// TIA Portal V19 export
FUNCTION_BLOCK "FB20_ManageState"   // FB20, LAD
{ S7_Optimized_Access := 'TRUE' }
// stored: AutoNumber false, IsIECCheckEnabled true, MemoryReserve 100, SetENOAutomatically false
   VAR_INPUT
      xGlobalSafety { ExternalAccessible := 'False'; ExternalVisible := 'False'; ExternalWritable := 'False'} : Bool;
      xGlobalFault { ExternalAccessible := 'False'; ExternalVisible := 'False'; ExternalWritable := 'False'} : Bool;
      xInformation { ExternalAccessible := 'False'; ExternalVisible := 'False'; ExternalWritable := 'False'} : Bool;
   END_VAR
   VAR_OUTPUT
      nGlobalState { ExternalAccessible := 'False'; ExternalVisible := 'False'; ExternalWritable := 'False'} : Int;
      xSafetyState { ExternalAccessible := 'False'; ExternalVisible := 'False'; ExternalWritable := 'False'} : Bool;
   END_VAR
BEGIN

REGION Network 1: Safety fault
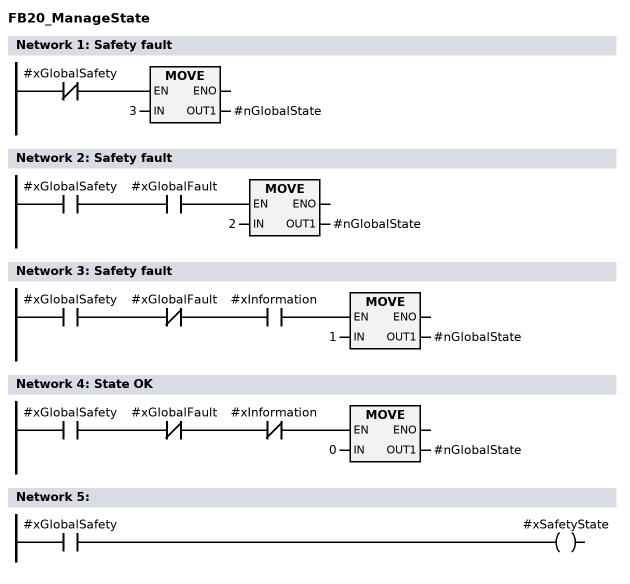
   RUNG wire#powerrail
      I_Contact( #xGlobalSafety )
      Move(in := 3, out1 => #nGlobalState)
   END_RUNG
   // the same network as SCL:
   IF NOT #xGlobalSafety THEN #nGlobalState := 3; END_IF;
END_REGION

REGION Network 2: Safety fault
   RUNG wire#powerrail
      Contact( #xGlobalSafety )
      Contact( #xGlobalFault )
      Move(in := 2, out1 => #nGlobalState)
   END_RUNG
   // the same network as SCL:
   IF #xGlobalSafety AND #xGlobalFault THEN #nGlobalState := 2; END_IF;
END_REGION

REGION Network 3: Safety fault
   RUNG wire#powerrail
      Contact( #xGlobalSafety )
      I_Contact( #xGlobalFault )
      Contact( #xInformation )
      Move(in := 1, out1 => #nGlobalState)
   END_RUNG
   // the same network as SCL:
   IF #xGlobalSafety AND NOT #xGlobalFault AND #xInformation THEN #nGlobalState := 1; END_IF;
END_REGION

REGION Network 4: State OK
   RUNG wire#powerrail
      Contact( #xGlobalSafety )
      I_Contact( #xGlobalFault )
      I_Contact( #xInformation )
      Move(in := 0, out1 => #nGlobalState)
   END_RUNG
   // the same network as SCL:
   IF #xGlobalSafety AND NOT #xGlobalFault AND NOT #xInformation THEN #nGlobalState := 0; END_IF;
END_REGION

REGION Network 5
   RUNG wire#powerrail
      Contact( #xGlobalSafety )
      Coil( #xSafetyState )
   END_RUNG
   // the same network as SCL:
   #xSafetyState := #xGlobalSafety;
END_REGION
END_FUNCTION_BLOCK
